# B&R Automation Studio project JXCP_PROFINET_project
Automation Studio 4.9.3.144 SP; technology packages: mappView 5.11.3

## Configuration Config1

CPU X20CP1382, AutomationRuntime A4.73, Build 4.1.2, Safety 0.0, Vc V4.72.0

### Task classes (Cpu.sw)
```
Cyclic#2 (cycle 10000 us, tolerance 10000 us):
  JXCP_Test <- Technology.JXCP_Test.prg
Binaries: udbdef, mvLoader, FWRules, TCData, sysconf, Role, User, iomap, ashwd, asfw, arconfig, ashwac, asnxdb1
Libraries: AsBrMath, rp_funcx, runtime, fileio, astime
```

### Hardware
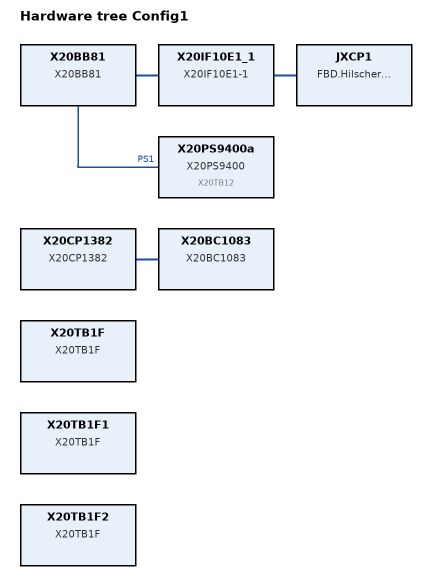
```
JXCP1 : FBD.Hilscher.PNIOGenDevDTM2.JXCP1 v0.0.0.0 (OrderNumber=JXCP1, VendorAddress=jxcp1)  [PN1 -> X20IF10E1_1.IF1]
  DtmId = 32d02dca-1395-427b-a27d-d5b2f34042f0
X20BB81 : X20BB81 v1.0.2.0
X20BC1083 : X20BC1083 v2.11.1.0  [PLK1 -> X20CP1382.IF3 [Cable Type=PowerlinkCable, Length=10, Version=1.0.0.3]; SL -> X20BB81.SL1]
X20CP1382 : X20CP1382 v1.11.0.0  [X1 -> X1.SL; X2 -> X2.SL; X3 -> X3.SL]
  Module X1 (Type=X1, Virtual=true, Version=1.11.0.0)
    Connection (Connector=SS1, TargetModule=X20TB1F, TargetConnector=SS)
    Connection (Connector=SL, TargetModule=X20CP1382, TargetConnector=X1)
  Module X2 (Type=X2, Virtual=true, Version=1.11.0.0)
    Connection (Connector=SS1, TargetModule=X20TB1F1, TargetConnector=SS)
    Connection (Connector=SL, TargetModule=X20CP1382, TargetConnector=X2)
  Module X3 (Type=X3, Virtual=true, Version=1.11.0.0)
    Connection (Connector=SS1, TargetModule=X20TB1F2, TargetConnector=SS)
    Connection (Connector=SL, TargetModule=X20CP1382, TargetConnector=X3)
  Connector IF2:
    ActivateDevice = 1
  Connector IF3:
    DNAConfiguration = manual
  ConfigurationID = JXCP_PROFINET_project_Config1
  Simulation = 1
  SystemTick = 2000
  TaskClassIdleTime = 2000
  Cyclic1Duration = 2000
  Cyclic1Tolerance = 0
  Cyclic2Duration = 10000
  Cyclic2Tolerance = 10000
  ActivateOpcUa = 1
  OpcUaInformationModels_PV_Version = 1
X20IF10E1_1 : X20IF10E1-1 v1.3.0.0  [SS -> X20BB81.SS1]
  Connector IF1:
    DtmRef = FBDIF.Hilscher.PNIOControllerDTM2.NETX 100 RE/PNM
    DtmId = 5926bdb0-bfe7-45dd-88e4-c4368abc1fd1
  ConfigFile = X20IF10E1_1.dtm
  ConfigModule = asnxdb1
  CycleTime = 2000
X20PS9400a : X20PS9400 v1.4.0.0  [SS1 -> X20TB12e.SS; PS -> X20BB81.PS1]
X20TB12e : X20TB12 v1.0.0.0
X20TB1F : X20TB1F v1.0.0.0
X20TB1F1 : X20TB1F v1.0.0.0
X20TB1F2 : X20TB1F v1.0.0.0
```

### IoMap.iom - X20CP1382/IoMap.iom
```iecst
VAR_CONFIG
	::JXCP_Test:jxcp_smc_fb_1.ModuleOK AT %IX."JXCP1".ModuleOk;
	::JXCP_Test.jxcp_smc_fb_1.PROFINET_Mapping_IN.Input_Area[0] AT %IB."JXCP1".Module001_IO_Input001;
	::JXCP_Test.jxcp_smc_fb_1.PROFINET_Mapping_IN.Input_Area[1] AT %IB."JXCP1".Module001_IO_Input002;
	::JXCP_Test.jxcp_smc_fb_1.PROFINET_Mapping_IN.Input_Area[2] AT %IB."JXCP1".Module001_IO_Input003;
	::JXCP_Test.jxcp_smc_fb_1.PROFINET_Mapping_IN.Input_Area[3] AT %IB."JXCP1".Module001_IO_Input004;
	::JXCP_Test.jxcp_smc_fb_1.PROFINET_Mapping_IN.Input_Area[4] AT %IB."JXCP1".Module001_IO_Input005;
	::JXCP_Test.jxcp_smc_fb_1.PROFINET_Mapping_IN.Input_Area[5] AT %IB."JXCP1".Module001_IO_Input006;
	::JXCP_Test.jxcp_smc_fb_1.PROFINET_Mapping_IN.Input_Area[6] AT %IB."JXCP1".Module001_IO_Input007;
	::JXCP_Test.jxcp_smc_fb_1.PROFINET_Mapping_IN.Input_Area[7] AT %IB."JXCP1".Module001_IO_Input008;
	::JXCP_Test.jxcp_smc_fb_1.PROFINET_Mapping_IN.Input_Area[8] AT %IB."JXCP1".Module001_IO_Input009;
	::JXCP_Test.jxcp_smc_fb_1.PROFINET_Mapping_IN.Input_Area[9] AT %IB."JXCP1".Module001_IO_Input010;
	::JXCP_Test.jxcp_smc_fb_1.PROFINET_Mapping_IN.Input_Area[10] AT %IB."JXCP1".Module001_IO_Input011;
	::JXCP_Test.jxcp_smc_fb_1.PROFINET_Mapping_IN.Input_Area[11] AT %IB."JXCP1".Module001_IO_Input012;
	::JXCP_Test.jxcp_smc_fb_1.PROFINET_Mapping_IN.Input_Area[12] AT %IB."JXCP1".Module001_IO_Input013;
	::JXCP_Test.jxcp_smc_fb_1.PROFINET_Mapping_IN.Input_Area[13] AT %IB."JXCP1".Module001_IO_Input014;
	::JXCP_Test.jxcp_smc_fb_1.PROFINET_Mapping_IN.Input_Area[14] AT %IB."JXCP1".Module001_IO_Input015;
	::JXCP_Test.jxcp_smc_fb_1.PROFINET_Mapping_IN.Input_Area[15] AT %IB."JXCP1".Module001_IO_Input016;
	::JXCP_Test.jxcp_smc_fb_1.PROFINET_Mapping_IN.Input_Area[16] AT %IB."JXCP1".Module001_IO_Input017;
	::JXCP_Test.jxcp_smc_fb_1.PROFINET_Mapping_IN.Input_Area[17] AT %IB."JXCP1".Module001_IO_Input018;
	::JXCP_Test.jxcp_smc_fb_1.PROFINET_Mapping_IN.Input_Area[18] AT %IB."JXCP1".Module001_IO_Input019;
	::JXCP_Test.jxcp_smc_fb_1.PROFINET_Mapping_IN.Input_Area[19] AT %IB."JXCP1".Module001_IO_Input020;
	::JXCP_Test:jxcp_smc_fb_1.PROFINET_Mapping_OUT.Output_Area[0] AT %QB."JXCP1".Module002_IO_Output001;
	::JXCP_Test:jxcp_smc_fb_1.PROFINET_Mapping_OUT.Output_Area[1] AT %QB."JXCP1".Module002_IO_Output002;
	::JXCP_Test:jxcp_smc_fb_1.PROFINET_Mapping_OUT.Output_Area[2] AT %QB."JXCP1".Module002_IO_Output003;
	::JXCP_Test:jxcp_smc_fb_1.PROFINET_Mapping_OUT.Output_Area[3] AT %QB."JXCP1".Module002_IO_Output004;
	::JXCP_Test:jxcp_smc_fb_1.PROFINET_Mapping_OUT.Output_Area[4] AT %QB."JXCP1".Module002_IO_Output005;
	::JXCP_Test:jxcp_smc_fb_1.PROFINET_Mapping_OUT.Output_Area[5] AT %QB."JXCP1".Module002_IO_Output006;
	::JXCP_Test:jxcp_smc_fb_1.PROFINET_Mapping_OUT.Output_Area[6] AT %QB."JXCP1".Module002_IO_Output007;
	::JXCP_Test:jxcp_smc_fb_1.PROFINET_Mapping_OUT.Output_Area[7] AT %QB."JXCP1".Module002_IO_Output008;
	::JXCP_Test:jxcp_smc_fb_1.PROFINET_Mapping_OUT.Output_Area[8] AT %QB."JXCP1".Module002_IO_Output009;
	::JXCP_Test:jxcp_smc_fb_1.PROFINET_Mapping_OUT.Output_Area[9] AT %QB."JXCP1".Module002_IO_Output010;
	::JXCP_Test:jxcp_smc_fb_1.PROFINET_Mapping_OUT.Output_Area[10] AT %QB."JXCP1".Module002_IO_Output011;
	::JXCP_Test:jxcp_smc_fb_1.PROFINET_Mapping_OUT.Output_Area[11] AT %QB."JXCP1".Module002_IO_Output012;
	::JXCP_Test:jxcp_smc_fb_1.PROFINET_Mapping_OUT.Output_Area[12] AT %QB."JXCP1".Module002_IO_Output013;
	::JXCP_Test:jxcp_smc_fb_1.PROFINET_Mapping_OUT.Output_Area[13] AT %QB."JXCP1".Module002_IO_Output014;
	::JXCP_Test:jxcp_smc_fb_1.PROFINET_Mapping_OUT.Output_Area[14] AT %QB."JXCP1".Module002_IO_Output015;
	::JXCP_Test:jxcp_smc_fb_1.PROFINET_Mapping_OUT.Output_Area[15] AT %QB."JXCP1".Module002_IO_Output016;
	::JXCP_Test:jxcp_smc_fb_1.PROFINET_Mapping_OUT.Output_Area[16] AT %QB."JXCP1".Module002_IO_Output017;
	::JXCP_Test:jxcp_smc_fb_1.PROFINET_Mapping_OUT.Output_Area[17] AT %QB."JXCP1".Module002_IO_Output018;
	::JXCP_Test:jxcp_smc_fb_1.PROFINET_Mapping_OUT.Output_Area[18] AT %QB."JXCP1".Module002_IO_Output019;
	::JXCP_Test:jxcp_smc_fb_1.PROFINET_Mapping_OUT.Output_Area[19] AT %QB."JXCP1".Module002_IO_Output020;
	::JXCP_Test:jxcp_smc_fb_1.PROFINET_Mapping_OUT.Output_Area[20] AT %QB."JXCP1".Module002_IO_Output021;
	::JXCP_Test:jxcp_smc_fb_1.PROFINET_Mapping_OUT.Output_Area[21] AT %QB."JXCP1".Module002_IO_Output022;
	::JXCP_Test:jxcp_smc_fb_1.PROFINET_Mapping_OUT.Output_Area[22] AT %QB."JXCP1".Module002_IO_Output023;
	::JXCP_Test:jxcp_smc_fb_1.PROFINET_Mapping_OUT.Output_Area[23] AT %QB."JXCP1".Module002_IO_Output024;
	::JXCP_Test:jxcp_smc_fb_1.PROFINET_Mapping_OUT.Output_Area[24] AT %QB."JXCP1".Module002_IO_Output025;
	::JXCP_Test:jxcp_smc_fb_1.PROFINET_Mapping_OUT.Output_Area[25] AT %QB."JXCP1".Module002_IO_Output026;
	::JXCP_Test:jxcp_smc_fb_1.PROFINET_Mapping_OUT.Output_Area[26] AT %QB."JXCP1".Module002_IO_Output027;
	::JXCP_Test:jxcp_smc_fb_1.PROFINET_Mapping_OUT.Output_Area[27] AT %QB."JXCP1".Module002_IO_Output028;
	::JXCP_Test:jxcp_smc_fb_1.PROFINET_Mapping_OUT.Output_Area[28] AT %QB."JXCP1".Module002_IO_Output029;
	::JXCP_Test:jxcp_smc_fb_1.PROFINET_Mapping_OUT.Output_Area[29] AT %QB."JXCP1".Module002_IO_Output030;
	::JXCP_Test:jxcp_smc_fb_1.PROFINET_Mapping_OUT.Output_Area[30] AT %QB."JXCP1".Module002_IO_Output031;
	::JXCP_Test:jxcp_smc_fb_1.PROFINET_Mapping_OUT.Output_Area[31] AT %QB."JXCP1".Module002_IO_Output032;
	::JXCP_Test:jxcp_smc_fb_1.PROFINET_Mapping_OUT.Output_Area[32] AT %QB."JXCP1".Module002_IO_Output033;
	::JXCP_Test:jxcp_smc_fb_1.PROFINET_Mapping_OUT.Output_Area[33] AT %QB."JXCP1".Module002_IO_Output034;
	::JXCP_Test:jxcp_smc_fb_1.PROFINET_Mapping_OUT.Output_Area[34] AT %QB."JXCP1".Module002_IO_Output035;
	::JXCP_Test:jxcp_smc_fb_1.PROFINET_Mapping_OUT.Output_Area[35] AT %QB."JXCP1".Module002_IO_Output036;
END_VAR
```

## Logical view

Binary libraries used (declarations not repeated): operator, runtime, astime, AsIecCon, AsBrMath

### Global.typ - Global data types
```iecst
TYPE
	jxcp_mv_alarm_str : 	STRUCT
		Alarm_1 : USINT;
		Alarm_1_img : BOOL;
		Alarm_2 : USINT;
		Alarm_2_img : BOOL;
		Alarm_3 : USINT;
		Alarm_3_img : BOOL;
		Alarm_4 : USINT;
		Alarm_4_img : BOOL;
	END_STRUCT;
	jxcp_mv_get_param_str : 	STRUCT
		Position : LREAL;
		Speed : LREAL;
		Force : LREAL;
		In_Pos : BOOL;
	END_STRUCT;
	jxcp_data_mv_str : 	STRUCT
		Power : BOOL;
		Home : BOOL;
		isHome : BOOL;
		PowerOn : BOOL;
		Control : jxcp_mv_control_str;
		Write_Parameters : jxcp_mv_set_param_str;
		Read_Parameters : jxcp_mv_get_param_str;
		Alarm : jxcp_mv_alarm_str;
		Reset_Alarm : BOOL;
	END_STRUCT;
	jxcp_mv_cm_str : 	STRUCT
		Start : BOOL;
		Stop : BOOL;
		Default_Param : BOOL;
	END_STRUCT;
	jxcp_mv_control_str : 	STRUCT
		Jog_pos : BOOL;
		Jog_neg : BOOL;
		Cycle_Mode : jxcp_mv_cm_str;
	END_STRUCT;
	jxcp_mv_set_param_str : 	STRUCT
		Position : LREAL;
		Speed : LREAL;
		Acceleration : LREAL;
		Deceleration : LREAL;
	END_STRUCT;
END_TYPE
```

### Global.var - Global variables
```iecst
VAR
	jxcp_data_mv : jxcp_data_mv_str;
END_VAR
```

### Package Logical/Libraries - Global libraries

### Library Logical/Libraries/rp_funcx (ANSIC)

#### Types.typ - Exported data types
```iecst
TYPE
	profinet_aux_m_str : 	STRUCT
		IN_Aux : profinet_aux_in_str;
		OUT_Aux : profinet_aux_out_str;
	END_STRUCT;
	profinet_aux_out_str : 	STRUCT
		BYTE_0 : ARRAY[0..5]OF BOOL;
		BYTE_1 : ARRAY[0..7]OF BOOL;
		BYTE_2 : BOOL;
	END_STRUCT;
	jxcp_main_read_enum :
		(
		JXCP_R_INITIALIZATION_STATE := 0,
		JXCP_R_RW_STATE := 10,
		JXCP_R_ERROR_MODE_STATE := 20
		);
	profinet_aux_in_str : 	STRUCT
		BYTE_0 : ARRAY[0..5]OF BOOL;
		BYTE_1 : ARRAY[0..7]OF BOOL;
		BYTE_2 : ARRAY[0..7]OF BOOL;
		BYTE_3 : ARRAY[0..7]OF BOOL;
	END_STRUCT;
	jxcp_main_enum :
		(
		JXCP_INITIALIZATION_STATE := 0,
		JXCP_WAIT_STATE := 10,
		JXCP_CYCLE_MODE_STATE := 20,
		JXCP_ALARM_MODE_STATE := 30,
		JXCP_ERROR_MODE_STATE := 40
		);
	set_param_mode_enum :
		(
		CYCLE_MOVE_MODE := 0
		);
	internal_param_str : 	STRUCT
		actual_state : jxcp_main_enum;
		before_state : jxcp_main_enum;
		actual_r_state : jxcp_main_read_enum;
		before_r_state : jxcp_main_read_enum;
		Profinet : profinet_aux_m_str;
	END_STRUCT;
	set_param_str : 	STRUCT
		Start : BOOL;
		Stop : BOOL;
		Mode : set_param_mode_enum;
		Boundary : boundary_str;
	END_STRUCT;
	byte_3_in_str : 	STRUCT
		Deceleration : BOOL;
		Pushing_Force : BOOL;
		Trigger_LV : BOOL;
		Pushing_Speed : BOOL;
		Moving_Force : BOOL;
		Area_out_1 : BOOL;
		Area_out_2 : BOOL;
		IN_Pos_Tolerance : BOOL;
	END_STRUCT;
	byte_2_in_str : 	STRUCT
		Speed_Restriction : BOOL;
		Movement_Mode : BOOL;
		Speed : BOOL;
		Position : BOOL;
		Acceleration : BOOL;
	END_STRUCT;
	byte_1_in_str : 	STRUCT
		HOLD : BOOL;
		SVON : BOOL;
		DRIVE : BOOL;
		RESET : BOOL;
		SETUP : BOOL;
		JOG_Neg : BOOL;
		JOG_Pos : BOOL;
		FLHGT : BOOL;
	END_STRUCT;
	byte_0_in_str : 	STRUCT
		IN_0 : BOOL;
		IN_1 : BOOL;
		IN_2 : BOOL;
		IN_3 : BOOL;
		IN_4 : BOOL;
		IN_5 : BOOL;
	END_STRUCT;
	movement_mode_str : 	STRUCT
		Absolute : BOOL;
		Relative : BOOL;
	END_STRUCT;
	alarm_str : 	STRUCT
		Alarm_1 : USINT;
		Alarm_2 : USINT;
		Alarm_3 : USINT;
		Alarm_4 : USINT;
	END_STRUCT;
	byte_2_str : 	STRUCT
		READY : BOOL;
	END_STRUCT;
	byte_1_str : 	STRUCT
		BUSY : BOOL;
		SVRE : BOOL;
		SETON : BOOL;
		INP : BOOL;
		AREA : BOOL;
		WAREA : BOOL;
		ESTOP : BOOL;
		ALARM : BOOL;
	END_STRUCT;
	byte_0_str : 	STRUCT
		OUT_0 : BOOL;
		OUT_1 : BOOL;
		OUT_2 : BOOL;
		OUT_3 : BOOL;
		OUT_4 : BOOL;
		OUT_5 : BOOL;
	END_STRUCT;
	jxcp_input_str : 	STRUCT
		BYTE_0 : byte_0_in_str;
		BYTE_1 : byte_1_in_str;
		BYTE_2 : byte_2_in_str;
		BYTE_3 : byte_3_in_str;
		Start_Flag : BOOL;
		Movement_Mode : movement_mode_str;
		Speed : LREAL;
		Position : LREAL;
		Acceleration : LREAL;
		Deceleration : LREAL;
		Pushing_Force : LREAL;
		Trigger_LV : LREAL;
		Pushing_Speed : LREAL;
		Moving_Force : LREAL;
		AREA_1 : LREAL;
		AREA_2 : LREAL;
		IN_Position : LREAL;
	END_STRUCT;
	jxcp_output_str : 	STRUCT
		BYTE_0 : byte_0_str;
		BYTE_1 : byte_1_str;
		BYTE_2 : byte_2_str;
		Current_Position : LREAL;
		Current_Speed : LREAL;
		Current_Pushing_Force : LREAL;
		Target_Position : LREAL;
		Warning : alarm_str;
	END_STRUCT;
	profinet_mapping_out_str : 	STRUCT
		Output_Area : ARRAY[0..35]OF USINT;
	END_STRUCT;
	profinet_mapping_in_str : 	STRUCT
		Input_Area : ARRAY[0..19]OF USINT;
	END_STRUCT;
	boundary_mm_str : 	STRUCT
		max : LREAL;
		min : LREAL;
	END_STRUCT;
	boundary_str : 	STRUCT
		Position : boundary_mm_str;
		Speed : boundary_mm_str;
		Acceleration : boundary_mm_str;
		Deceleration : boundary_mm_str;
	END_STRUCT;
END_TYPE
```

#### rp_funcx.fun - Exported functions and function blocks
```iecst
FUNCTION_BLOCK dec_to_multiple_usint
	VAR_INPUT
		Count_of_VAR : USINT;
		Decimal : LREAL;
	END_VAR
	VAR_OUTPUT
		Result_USINT_1 : USINT;
		Result_USINT_2 : USINT;
		Result_USINT_3 : USINT;
		Result_USINT_4 : USINT;
	END_VAR
END_FUNCTION_BLOCK

FUNCTION_BLOCK multiplne_usint_to_dec
	VAR_INPUT
		Count_of_VAR : USINT;
		USINT_1 : USINT;
		USINT_2 : USINT;
		USINT_3 : USINT;
		USINT_4 : USINT;
	END_VAR
	VAR_OUTPUT
		Result_Decimal : LREAL;
	END_VAR
END_FUNCTION_BLOCK

{REDUND_ERROR} FUNCTION_BLOCK jxcp_smc_fb (*TODO: Add your comment here*) (*$GROUP=User,$CAT=User,$GROUPICON=User.png,$CATICON=User.png*)
	VAR_INPUT
		Enable : {REDUND_UNREPLICABLE} BOOL;
		ModuleOK : BOOL;
		PROFINET_Mapping_IN : {REDUND_UNREPLICABLE} profinet_mapping_in_str;
		Input : jxcp_input_str;
		Set_Parameters : set_param_str;
	END_VAR
	VAR_OUTPUT
		Active : BOOL;
		PROFINET_Mapping_OUT : profinet_mapping_out_str;
		Output : jxcp_output_str;
	END_VAR
	VAR
		Internal : internal_param_str;
	END_VAR
END_FUNCTION_BLOCK
```

#### jxcp_smc_fb.c
```c
// ************************************************************************************************************************************ //
// Title: JXCP1 (SMC) - Control {PROFINET}
// Autor: Roman Parak
// Date : 8.5.2020
// Email: Roman.Parak@outlook.com
// ************************************************************************************************************************************ //

// ************************************************************************************************************************************ //
// -------------------------------------------------------------  LIBRARIES ----------------------------------------------------------- //
// ************************************************************************************************************************************ //
#include <bur/plctypes.h>
#include <stdio.h>
#include <stdlib.h>
#include <math.h>

#ifdef __cplusplus
	extern "C"
	{
#endif
#include "rp_funcx.h"
#ifdef __cplusplus
	};
#endif

// ************************************************************************************************************************************ //
// -------------------------------------------------------------  DECLARATIONS -------------------------------------------------------- //
// ************************************************************************************************************************************ //
// INITIALIZATION // RESET //
void initialization_jxcp(struct jxcp_smc_fb* jxcp_s);

// INITIALIZATION // AUX. FCE. Convert Binary to Decimal //
DINT convert_bin_to_dec(LREAL n);

// ************************************************************************************************************************************ //
// --------------------------------------------------------------  MAIN --------------------------------------------------------------- //
// ************************************************************************************************************************************ //
void jxcp_smc_fb(struct jxcp_smc_fb* jxcp_s)
{
	// *********************************************************//
	// ---------------- INITIALIZATION  ----------------------- //
	// *********************************************************//
	if(jxcp_s->Enable != 1){
		initialization_jxcp(jxcp_s);
	}

	// declaration index {all cycles)
	int i, i_w;

	// Read {Multiple USINT to Decimal -> Function Block}
	struct multiple_usint_to_dec m_u2d_cP; // Current Position
	struct multiple_usint_to_dec m_u2d_cS; // Current Speed
	struct multiple_usint_to_dec m_u2d_cPF; // Current Pushing Force
	struct multiple_usint_to_dec m_u2d_TP; // Target Position

	// Write {Decimal to multiple USINT -> Function Block}
	struct dec_to_multiple_usint dec2u_m_S; // Speed
	struct dec_to_multiple_usint dec2u_m_P; // Position
	struct dec_to_multiple_usint dec2u_m_Acc; // Acceleration
	struct dec_to_multiple_usint dec2u_m_Dec; // Deceleration
	struct dec_to_multiple_usint dec2u_m_PF; // Pushing Force
	struct dec_to_multiple_usint dec2u_m_TLV; // Trigger LV
	struct dec_to_multiple_usint dec2u_m_PS; // Pushing Speed
	struct dec_to_multiple_usint dec2u_m_MF; // Moving FOrce
	struct dec_to_multiple_usint dec2u_m_AR1; // Area 1
	struct dec_to_multiple_usint dec2u_m_AR2; // Area 2
	struct dec_to_multiple_usint dec2u_m_IN_P; // IN Position

	// ******************************************************************************************************************//
	// --------------------------------------------- JXCP MAIN STATE  -------------------------------------------------- //
	// ******************************************************************************************************************//
	switch(jxcp_s->Internal.actual_state){
		case JXCP_INITIALIZATION_STATE:
			{
				/*************************************** INITIALIZATION STATE ******************************************/
				jxcp_s->Internal.before_state = JXCP_INITIALIZATION_STATE;
				// Profinet Module -> OK
				if(jxcp_s->ModuleOK == 1){
					// Set FB -> Active 1
					jxcp_s->Active = 1;
					// Change State -> Wait
					jxcp_s->Internal.actual_state = JXCP_WAIT_STATE;
				}
			}
			break;
		case JXCP_WAIT_STATE:
			{
				/*************************************** WAIT STATE ******************************************/
				jxcp_s->Internal.before_state = JXCP_WAIT_STATE;

				jxcp_s->Set_Parameters.Stop = 0;

				// *************** Start Mode *************** //
				if(jxcp_s->Set_Parameters.Start == 1){
					if(jxcp_s->Set_Parameters.Mode == NORMAL_MOVE_MODE){
						// Normal Mode
						jxcp_s->Internal.actual_state = JXCP_NORMAL_MODE_STATE;
					}else if(jxcp_s->Set_Parameters.Mode == CYCLE_MOVE_MODE){
						// Write Byte 2 { SET - 1 }
						jxcp_s->Input.BYTE_2.Speed_Restriction = 1;
						jxcp_s->Input.BYTE_2.Movement_Mode     = 1;
						jxcp_s->Input.BYTE_2.Speed             = 1;
						jxcp_s->Input.BYTE_2.Position          = 1;
						jxcp_s->Input.BYTE_2.Acceleration      = 1;
						// Write Byte 3 { SET - 1 }
						jxcp_s->Input.BYTE_3.Deceleration      = 1;
						jxcp_s->Input.BYTE_3.Pushing_Force     = 1;
						jxcp_s->Input.BYTE_3.Trigger_LV        = 1;
						jxcp_s->Input.BYTE_3.Pushing_Speed     = 1;
						jxcp_s->Input.BYTE_3.Moving_Force      = 1;
						jxcp_s->Input.BYTE_3.Area_out_1        = 1;
						jxcp_s->Input.BYTE_3.Area_out_2        = 1;
						jxcp_s->Input.BYTE_3.IN_Pos_Tolerance  = 1;
						// Cycle Mode
						jxcp_s->Internal.actual_state = JXCP_CYCLE_MODE_STATE;
					}
				}

				// Module OK = 0 -> Error State
				if(jxcp_s->ModuleOK != 1){
					// Set FB -> Active 0
					jxcp_s->Active = 0;
					// Change State -> Error
					jxcp_s->Internal.actual_state = JXCP_ERROR_MODE_STATE;
				}
			}
			break;
		case JXCP_NORMAL_MODE_STATE:
			{
				/*************************************** NORMAL MODE STATE ******************************************/
				jxcp_s->Internal.before_state = JXCP_NORMAL_MODE_STATE;

				// *************** Stop Actual Mode *************** //
				if(jxcp_s->Set_Parameters.Stop == 1){
					jxcp_s->Set_Parameters.Start = 0;
					// Change State -> Initialization
					jxcp_s->Internal.actual_state = JXCP_WAIT_STATE;
				}

				// Module OK = 0 -> Error State
				if(jxcp_s->ModuleOK != 1){
					// Set FB -> Active 0
					jxcp_s->Active = 0;
					// Change State -> Error
					jxcp_s->Internal.actual_state = JXCP_ERROR_MODE_STATE;
				}
			}
			break;
		case JXCP_CYCLE_MODE_STATE:
			{
				/*************************************** CYCLE MODE STATE ******************************************/
				jxcp_s->Internal.before_state = JXCP_CYCLE_MODE_STATE;

				// Start Cycle Mode -> JXCP1 command
				jxcp_s->Input.Start_Flag 			 = 1;
				// Movement Mode - Absolute
				jxcp_s->Input.Movement_Mode.Absolute = 1;

				/*************************************************************************/
				/*************** Calculation  DEC. TO MULTIPLE USINT *********************/
				/*************************************************************************/

				// *************** Speed *************** //
				// Number of Variables (USINT)
				dec2u_m_S.Count_of_VAR = 2;
				// Boundary Condition
				if(jxcp_s->Input.Speed > jxcp_s->Set_Parameters.Boundary.Speed.max){
					dec2u_m_S.Decimal = jxcp_s->Set_Parameters.Boundary.Speed.max;
				}else if(jxcp_s->Input.Speed < jxcp_s->Set_Parameters.Boundary.Speed.min){
					dec2u_m_S.Decimal = jxcp_s->Set_Parameters.Boundary.Speed.min;
				}else{
					dec2u_m_S.Decimal = jxcp_s->Input.Speed;
				}
				// Call Function Block (Decimal to Multiple USINT)
				dec_to_multiple_usint(&dec2u_m_S);
				// Result (Write -> PROFINET Module)
				jxcp_s->PROFINET_Mapping_OUT.Output_Area[6] = dec2u_m_S.Result_USINT_1;
				jxcp_s->PROFINET_Mapping_OUT.Output_Area[7] = dec2u_m_S.Result_USINT_2;

				// *************** Position *************** //
				// Number of Variables (USINT)
				dec2u_m_P.Count_of_VAR = 4;
				// Boundary Condition
				if(jxcp_s->Input.Position > jxcp_s->Set_Parameters.Boundary.Position.max){
					dec2u_m_P.Decimal = jxcp_s->Set_Parameters.Boundary.Position.max;
				}else if(jxcp_s->Input.Position < jxcp_s->Set_Parameters.Boundary.Position.min){
					dec2u_m_P.Decimal = jxcp_s->Set_Parameters.Boundary.Position.min;
				}else{
					dec2u_m_P.Decimal = jxcp_s->Input.Position;
				}
				// Call Function Block (Decimal to Multiple USINT)
				dec_to_multiple_usint(&dec2u_m_P);
				// Result (Write -> PROFINET Module)
				jxcp_s->PROFINET_Mapping_OUT.Output_Area[8] = dec2u_m_P.Result_USINT_1;
				jxcp_s->PROFINET_Mapping_OUT.Output_Area[9] = dec2u_m_P.Result_USINT_2;
				jxcp_s->PROFINET_Mapping_OUT.Output_Area[10] = dec2u_m_P.Result_USINT_3;
				jxcp_s->PROFINET_Mapping_OUT.Output_Area[11] = dec2u_m_P.Result_USINT_4;

				// *************** Acceleration *************** //
				// Number of Variables (USINT)
				dec2u_m_Acc.Count_of_VAR = 2;
				// Boundary Condition
				if(jxcp_s->Input.Acceleration > jxcp_s->Set_Parameters.Boundary.Acceleration.max){
					dec2u_m_Acc.Decimal = jxcp_s->Set_Parameters.Boundary.Acceleration.max;
				}else if(jxcp_s->Input.Acceleration < jxcp_s->Set_Parameters.Boundary.Acceleration.min){
					dec2u_m_Acc.Decimal = jxcp_s->Set_Parameters.Boundary.Acceleration.min;
				}else{
					dec2u_m_Acc.Decimal = jxcp_s->Input.Acceleration;
				}
				// Call Function Block (Decimal to Multiple USINT)
				dec_to_multiple_usint(&dec2u_m_Acc);
				// Result (Write -> PROFINET Module)
				jxcp_s->PROFINET_Mapping_OUT.Output_Area[12] = dec2u_m_Acc.Result_USINT_1;
				jxcp_s->PROFINET_Mapping_OUT.Output_Area[13] = dec2u_m_Acc.Result_USINT_2;

				// *************** Deceleration *************** //
				// Number of Variables (USINT)
				dec2u_m_Dec.Count_of_VAR = 2;
				// Boundary Condition
				if(jxcp_s->Input.Deceleration > jxcp_s->Set_Parameters.Boundary.Deceleration.max){
					dec2u_m_Dec.Decimal = jxcp_s->Set_Parameters.Boundary.Deceleration.max;
				}else if(jxcp_s->Input.Deceleration < jxcp_s->Set_Parameters.Boundary.Deceleration.min){
					dec2u_m_Dec.Decimal = jxcp_s->Set_Parameters.Boundary.Deceleration.min;
				}else{
					dec2u_m_Dec.Decimal = jxcp_s->Input.Deceleration;
				}
				// Call Function Block (Decimal to Multiple USINT)
				dec_to_multiple_usint(&dec2u_m_Dec);
				// Result (Write -> PROFINET Module)
				jxcp_s->PROFINET_Mapping_OUT.Output_Area[14] = dec2u_m_Dec.Result_USINT_1;
				jxcp_s->PROFINET_Mapping_OUT.Output_Area[15] = dec2u_m_Dec.Result_USINT_2;

				// *************** Pushing Force *************** //
				// Number of Variables (USINT)
				dec2u_m_PF.Count_of_VAR = 2;
				// Boundary Condition (NO)
				dec2u_m_PF.Decimal = jxcp_s->Input.Pushing_Force;
				// Call Function Block (Decimal to Multiple USINT)
				dec_to_multiple_usint(&dec2u_m_PF);
				// Result (Write -> PROFINET Module)
				jxcp_s->PROFINET_Mapping_OUT.Output_Area[16] = dec2u_m_PF.Result_USINT_1;
				jxcp_s->PROFINET_Mapping_OUT.Output_Area[17] = dec2u_m_PF.Result_USINT_2;

				// *************** Trigger LV *************** //
				// Number of Variables (USINT)
				dec2u_m_TLV.Count_of_VAR = 2;
				// Boundary Condition (NO)
				dec2u_m_TLV.Decimal = jxcp_s->Input.Trigger_LV;
				// Call Function Block (Decimal to Multiple USINT)
				dec_to_multiple_usint(&dec2u_m_TLV);
				// Result (Write -> PROFINET Module)
				jxcp_s->PROFINET_Mapping_OUT.Output_Area[18] = dec2u_m_TLV.Result_USINT_1;
				jxcp_s->PROFINET_Mapping_OUT.Output_Area[19] = dec2u_m_TLV.Result_USINT_2;

				// *************** Pushing Speed *************** //
				// Number of Variables (USINT)
				dec2u_m_PS.Count_of_VAR = 2;
				// Boundary Condition (NO)
				dec2u_m_PS.Decimal = jxcp_s->Input.Pushing_Speed;
				// Call Function Block (Decimal to Multiple USINT)
				dec_to_multiple_usint(&dec2u_m_PS);
				// Result (Write -> PROFINET Module)
				jxcp_s->PROFINET_Mapping_OUT.Output_Area[20] = dec2u_m_PS.Result_USINT_1;
				jxcp_s->PROFINET_Mapping_OUT.Output_Area[21] = dec2u_m_PS.Result_USINT_2;

				// *************** Moving Force *************** //
				// Number of Variables (USINT)
				dec2u_m_MF.Count_of_VAR = 2;
				// Boundary Condition (NO)
				dec2u_m_MF.Decimal = jxcp_s->Input.Moving_Force;
				// Call Function Block (Decimal to Multiple USINT)
				dec_to_multiple_usint(&dec2u_m_MF);
				// Result (Write -> PROFINET Module)
				jxcp_s->PROFINET_Mapping_OUT.Output_Area[22] = dec2u_m_MF.Result_USINT_1;
				jxcp_s->PROFINET_Mapping_OUT.Output_Area[23] = dec2u_m_MF.Result_USINT_2;

				// *************** Area 1 *************** //
				// Number of Variables (USINT)
				dec2u_m_AR1.Count_of_VAR = 4;
				// Boundary Condition (NO)
				dec2u_m_AR1.Decimal = jxcp_s->Input.AREA_1;
				// Call Function Block (Decimal to Multiple USINT)
				dec_to_multiple_usint(&dec2u_m_AR1);
				// Result (Write -> PROFINET Module)
				jxcp_s->PROFINET_Mapping_OUT.Output_Area[24] = dec2u_m_AR1.Result_USINT_1;
				jxcp_s->PROFINET_Mapping_OUT.Output_Area[25] = dec2u_m_AR1.Result_USINT_2;
				jxcp_s->PROFINET_Mapping_OUT.Output_Area[26] = dec2u_m_AR1.Result_USINT_3;
				jxcp_s->PROFINET_Mapping_OUT.Output_Area[27] = dec2u_m_AR1.Result_USINT_4;

				// *************** Area 2 *************** //
				// Number of Variables (USINT)
				dec2u_m_AR2.Count_of_VAR = 4;
				// Boundary Condition (NO)
				dec2u_m_AR2.Decimal = jxcp_s->Input.AREA_2;
				// Call Function Block (Decimal to Multiple USINT)
				dec_to_multiple_usint(&dec2u_m_AR2);
				// Result (Write -> PROFINET Module)
				jxcp_s->PROFINET_Mapping_OUT.Output_Area[28] = dec2u_m_AR2.Result_USINT_1;
				jxcp_s->PROFINET_Mapping_OUT.Output_Area[29] = dec2u_m_AR2.Result_USINT_2;
				jxcp_s->PROFINET_Mapping_OUT.Output_Area[30] = dec2u_m_AR2.Result_USINT_3;
				jxcp_s->PROFINET_Mapping_OUT.Output_Area[31] = dec2u_m_AR2.Result_USINT_4;

				// *************** In-Position *************** //
				// Number of Variables (USINT)
				dec2u_m_IN_P.Count_of_VAR = 4;
				// Boundary Condition (NO)
				dec2u_m_IN_P.Decimal = jxcp_s->Input.IN_Position;
				// Call Function Block (Decimal to Multiple USINT)
				dec_to_multiple_usint(&dec2u_m_IN_P);
				// Result (Write -> PROFINET Module)
				jxcp_s->PROFINET_Mapping_OUT.Output_Area[32] = dec2u_m_IN_P.Result_USINT_1;
				jxcp_s->PROFINET_Mapping_OUT.Output_Area[33] = dec2u_m_IN_P.Result_USINT_2;
				jxcp_s->PROFINET_Mapping_OUT.Output_Area[34] = dec2u_m_IN_P.Result_USINT_3;
				jxcp_s->PROFINET_Mapping_OUT.Output_Area[35] = dec2u_m_IN_P.Result_USINT_4;

				// *************** Stop Actual Mode *************** //
				if(jxcp_s->Set_Parameters.Stop == 1){
					jxcp_s->Set_Parameters.Start = 0;
					// Write Byte 4 { SET - 0 }
					jxcp_s->Input.Start_Flag 			   = 0;
					// Write Byte 2 { SET - 0 }
					jxcp_s->Input.BYTE_2.Speed_Restriction = 0;
					jxcp_s->Input.BYTE_2.Movement_Mode     = 0;
					jxcp_s->Input.BYTE_2.Speed             = 0;
					jxcp_s->Input.BYTE_2.Position          = 0;
					jxcp_s->Input.BYTE_2.Acceleration      = 0;
					// Write Byte 3 { SET - 0 }
					jxcp_s->Input.BYTE_3.Deceleration      = 0;
					jxcp_s->Input.BYTE_3.Pushing_Force     = 0;
					jxcp_s->Input.BYTE_3.Trigger_LV        = 0;
					jxcp_s->Input.BYTE_3.Pushing_Speed     = 0;
					jxcp_s->Input.BYTE_3.Moving_Force      = 0;
					jxcp_s->Input.BYTE_3.Area_out_1        = 0;
					jxcp_s->Input.BYTE_3.Area_out_2        = 0;
					jxcp_s->Input.BYTE_3.IN_Pos_Tolerance  = 0;
					// Change State -> Initialization
					jxcp_s->Internal.actual_state = JXCP_WAIT_STATE;
				}

				// Module OK = 0 -> Error State
				if(jxcp_s->ModuleOK != 1){
					// Set FB -> Active 0
					jxcp_s->Active = 0;
					// Change State -> Error
					jxcp_s->Internal.actual_state = JXCP_ERROR_MODE_STATE;
				}
			}
			break;
		case JXCP_ALARM_MODE_STATE:
			{
				/*************************************** ALARM STATE ******************************************/
				jxcp_s->Internal.before_state = JXCP_ALARM_MODE_STATE;

				// Module OK = 0 -> Error State
				if(jxcp_s->ModuleOK != 1){
					// Set FB -> Active 0
					jxcp_s->Active = 0;
					// Change State -> Error
					jxcp_s->Internal.actual_state = JXCP_ERROR_MODE_STATE;
				}
			}
			break;
		case JXCP_ERROR_MODE_STATE:
			{
				/*************************************** ERROR STATE ******************************************/
				// Profinet Module -> OK
				if(jxcp_s->ModuleOK == 1){
					// Set FB -> Active 1
					jxcp_s->Active = 1;
					// Change State -> before state (before the error)
					jxcp_s->Internal.actual_state = jxcp_s->Internal.before_state;
				}
			}
			break;
	} // end switch

	// ******************************************************************************************************************//
	// ---------------------------------------------------- JXCP R/W STATE  -------------------------------------------- //
	// ******************************************************************************************************************//
	switch(jxcp_s->Internal.actual_r_state){
		case JXCP_R_INITIALIZATION_STATE:
			{
				/*************************************** INITIALIZATION STATE ******************************************/
				jxcp_s->Internal.before_r_state = JXCP_R_INITIALIZATION_STATE;
				// Profinet Module -> OK
				if(jxcp_s->ModuleOK == 1){
					// Set FB -> Active
					jxcp_s->Active = 1;
					// Change State -> Read/Write
					jxcp_s->Internal.actual_r_state = JXCP_R_RW_STATE;
				}
			}
			break;
		case JXCP_R_RW_STATE:
			{
				/*************************************** READ/WRITE STATE ******************************************/
				jxcp_s->Internal.before_r_state = JXCP_R_RW_STATE;

				// ************************************************************************ //
				// ********************************* READ ********************************* //
				// ************************************************************************ //

				// *************** Byte 0 *************** //
				// Create aux. variable
				USINT aux_get_byte_0;
				// Read Profinet Var.
				aux_get_byte_0 = jxcp_s->PROFINET_Mapping_IN.Input_Area[0];
				// Calculation Boolean (True/False) array (Byte 0)
				for(i = 0; i < (int)(sizeof(jxcp_s->Internal.Profinet.OUT_Aux.BYTE_0)/sizeof(jxcp_s->Internal.Profinet.OUT_Aux.BYTE_0[0])); i++){
					if(aux_get_byte_0 > 0){
						jxcp_s->Internal.Profinet.OUT_Aux.BYTE_0[i] = aux_get_byte_0 % 2;
						aux_get_byte_0 = aux_get_byte_0/2;
					}else{
						jxcp_s->Internal.Profinet.OUT_Aux.BYTE_0[i] = 0;
					}
				}

				// *************** Byte 1 *************** //
				// Create aux. variable
				USINT aux_get_byte_1;
				// Read Profinet Var.
				aux_get_byte_1 = jxcp_s->PROFINET_Mapping_IN.Input_Area[1];
				// Calculation Boolean (True/False) array (Byte 1)
				for(i = 0; i < (int)(sizeof(jxcp_s->Internal.Profinet.OUT_Aux.BYTE_1)/sizeof(jxcp_s->Internal.Profinet.OUT_Aux.BYTE_1[0])); i++){
					if(aux_get_byte_1 > 0){
						jxcp_s->Internal.Profinet.OUT_Aux.BYTE_1[i] = aux_get_byte_1 % 2;
						aux_get_byte_1 = aux_get_byte_1/2;
					}else{
						jxcp_s->Internal.Profinet.OUT_Aux.BYTE_1[i] = 0;
					}
				}

				// *************** Byte 2 *************** //
				// Read Profinet Var. -> Set Bool
				if(jxcp_s->PROFINET_Mapping_IN.Input_Area[2] == 16){
					jxcp_s->Internal.Profinet.OUT_Aux.BYTE_2 = 1;
				}else{
					jxcp_s->Internal.Profinet.OUT_Aux.BYTE_2 = 0;
				}

				// *************** Current Position *************** //
				// Number of Variables (USINT)
				m_u2d_cP.Count_of_VAR = 4;
				// Read -> PROFINET Var.
				m_u2d_cP.USINT_1 = jxcp_s->PROFINET_Mapping_IN.Input_Area[4];
				m_u2d_cP.USINT_2 = jxcp_s->PROFINET_Mapping_IN.Input_Area[5];
				m_u2d_cP.USINT_3 = jxcp_s->PROFINET_Mapping_IN.Input_Area[6];
				m_u2d_cP.USINT_4 = jxcp_s->PROFINET_Mapping_IN.Input_Area[7];
				// Call Function Block (Multiple USINT to Decimal)
				multiple_usint_to_dec(&m_u2d_cP);
				// Result (Decimal Variable)
				jxcp_s->Output.Current_Position = m_u2d_cP.Result_Decimal;

				// *************** Current Speed *************** //
				// Number of Variables (USINT)
				m_u2d_cS.Count_of_VAR = 2;
				// Read -> PROFINET Var.
				m_u2d_cS.USINT_1 = jxcp_s->PROFINET_Mapping_IN.Input_Area[8];
				m_u2d_cS.USINT_2 = jxcp_s->PROFINET_Mapping_IN.Input_Area[9];
				// Call Function Block (Multiple USINT to Decimal)
				multiple_usint_to_dec(&m_u2d_cS);
				// Result (Decimal Variable)
				jxcp_s->Output.Current_Speed = m_u2d_cS.Result_Decimal;

				// *************** Current Pushing Force *************** //
				// Number of Variables (USINT)
				m_u2d_cPF.Count_of_VAR = 2;
				// Read -> PROFINET Var.
				m_u2d_cPF.USINT_1 = jxcp_s->PROFINET_Mapping_IN.Input_Area[10];
				m_u2d_cPF.USINT_2 = jxcp_s->PROFINET_Mapping_IN.Input_Area[11];
				// Call Function Block (Multiple USINT to Decimal)
				multiple_usint_to_dec(&m_u2d_cPF);
				// Result (Decimal Variable)
				jxcp_s->Output.Current_Pushing_Force = m_u2d_cPF.Result_Decimal;

				// *************** Target Position *************** //
				// Number of Variables (USINT)
				m_u2d_TP.Count_of_VAR = 4;
				// Read -> PROFINET Var.
				m_u2d_TP.USINT_1 = jxcp_s->PROFINET_Mapping_IN.Input_Area[12];
				m_u2d_TP.USINT_2 = jxcp_s->PROFINET_Mapping_IN.Input_Area[13];
				m_u2d_TP.USINT_3 = jxcp_s->PROFINET_Mapping_IN.Input_Area[14];
				m_u2d_TP.USINT_4 = jxcp_s->PROFINET_Mapping_IN.Input_Area[15];
				// Call Function Block (Multiple USINT to Decimal)
				multiple_usint_to_dec(&m_u2d_TP);
				// Result (Decimal Variable)
				jxcp_s->Output.Target_Position = m_u2d_TP.Result_Decimal;

				// *************** Byte 16 - 19 {ALARM} *************** //
				// Read -> PROFINET Var.
				jxcp_s->Output.Warning.Alarm_1 = jxcp_s->PROFINET_Mapping_IN.Input_Area[16];
				// Read -> PROFINET Var.
				jxcp_s->Output.Warning.Alarm_2 = jxcp_s->PROFINET_Mapping_IN.Input_Area[17];
				// Read -> PROFINET Var.
				jxcp_s->Output.Warning.Alarm_3 = jxcp_s->PROFINET_Mapping_IN.Input_Area[18];
				// Read -> PROFINET Var.
				jxcp_s->Output.Warning.Alarm_4 = jxcp_s->PROFINET_Mapping_IN.Input_Area[19];

				// ************************************************************************ //
				// ********************************* WRITE ******************************** //
				// ************************************************************************ //

				// *************** Byte 0 *************** //
				// Create aux. variable
				USINT aux_set_byte_0;
				// Initialization
				aux_set_byte_0 = 0;
				// Calculation from Boolean (True/False) -> USINT (Byte 0)
				for(i = 0; i < (int)(sizeof(jxcp_s->Internal.Profinet.IN_Aux.BYTE_0)/sizeof(jxcp_s->Internal.Profinet.IN_Aux.BYTE_0[0])); i++){
					if(jxcp_s->Internal.Profinet.IN_Aux.BYTE_0[i] == 1){
						aux_set_byte_0 += pow(2, i);
					}
				}
				// Result Profinet (USINT)
				jxcp_s->PROFINET_Mapping_OUT.Output_Area[0] = aux_set_byte_0;

				// *************** Byte 1 *************** //
				// Create aux. variable
				USINT aux_set_byte_1;
				// Initialization
				aux_set_byte_1 = 0;
				// Calculation from Boolean (True/False) -> USINT (Byte 1)
				for(i = 0; i < (int)(sizeof(jxcp_s->Internal.Profinet.IN_Aux.BYTE_1)/sizeof(jxcp_s->Internal.Profinet.IN_Aux.BYTE_1[0])); i++){
					if(jxcp_s->Internal.Profinet.IN_Aux.BYTE_1[i] == 1){
						aux_set_byte_1 += pow(2, i);
					}
				}
				// Result Profinet (USINT)
				jxcp_s->PROFINET_Mapping_OUT.Output_Area[1] = aux_set_byte_1;

				// *************** Byte 2 *************** //
				// Create aux. variable
				USINT aux_set_byte_2;
				// Initialization
				aux_set_byte_2 = 0;
				// Calculation from Boolean (True/False) -> USINT (Byte 2)
				for(i = 0; i < (int)(sizeof(jxcp_s->Internal.Profinet.IN_Aux.BYTE_2)/sizeof(jxcp_s->Internal.Profinet.IN_Aux.BYTE_2[0])); i++){
					if(jxcp_s->Internal.Profinet.IN_Aux.BYTE_2[i] == 1){
						aux_set_byte_2 += pow(2, i);
					}
				}
				// Result Profinet (USINT)
				jxcp_s->PROFINET_Mapping_OUT.Output_Area[2] = aux_set_byte_2;

				// *************** Byte 3 *************** //
				// Create aux. variable
				USINT aux_set_byte_3;
				// Initialization
				aux_set_byte_3 = 0;

				for(i = 0; i < (int)(sizeof(jxcp_s->Internal.Profinet.IN_Aux.BYTE_3)/sizeof(jxcp_s->Internal.Profinet.IN_Aux.BYTE_3[0])); i++){
					if(jxcp_s->Internal.Profinet.IN_Aux.BYTE_3[i] == 1){
						aux_set_byte_3 += pow(2, i);
					}
				}
				// Result Profinet (USINT)
				jxcp_s->PROFINET_Mapping_OUT.Output_Area[3] = aux_set_byte_3;

				// *************** Byte 4 *************** //
				// Write Profinet Var. -> Set USINT
				if(jxcp_s->Input.Start_Flag == 1){
					jxcp_s->PROFINET_Mapping_OUT.Output_Area[4] = 1;
				}else{
					jxcp_s->PROFINET_Mapping_OUT.Output_Area[4] = 0;
				}
				// *************** Byte 5 *************** //
				// Write Profinet Var. -> Set USINT
				if(jxcp_s->Input.Movement_Mode.Absolute == 1){
					// Movement -> Absolute
					jxcp_s->PROFINET_Mapping_OUT.Output_Area[5] = 1;
				}else if(jxcp_s->Input.Movement_Mode.Relative == 1){
					// Movement -> Relative
					jxcp_s->PROFINET_Mapping_OUT.Output_Area[5] = 2;
				}else{
					// Movement -> NULL
					jxcp_s->PROFINET_Mapping_OUT.Output_Area[5] = 0;
				}

				// Module OK = 0 -> Error State
				if(jxcp_s->ModuleOK != 1){
					// Set FB -> Active 0
					jxcp_s->Active = 0;
					// Change State -> Error
					jxcp_s->Internal.actual_r_state = JXCP_R_ERROR_MODE_STATE;
				}
			}
			break;
		case JXCP_R_ERROR_MODE_STATE:
			{
				/*************************************** ERROR STATE ******************************************/
				// Profinet Module -> OK
				if(jxcp_s->ModuleOK == 1){
					// Set FB -> Active 1
					jxcp_s->Active = 1;
					// Change State -> before state (before the error)
					jxcp_s->Internal.actual_r_state = jxcp_s->Internal.before_r_state;
				}
			}
			break;
	} // end switch

	/*************************************** R/W DATA ******************************************/
	if(jxcp_s->Active == 1){
		// Read Data {Transform Single Data -> ARRAY}
		// Byte 0 {INPUT}
		jxcp_s->Internal.Profinet.IN_Aux.BYTE_0[0] = jxcp_s->Input.BYTE_0.IN_0;
		jxcp_s->Internal.Profinet.IN_Aux.BYTE_0[1] = jxcp_s->Input.BYTE_0.IN_1;
		jxcp_s->Internal.Profinet.IN_Aux.BYTE_0[2] = jxcp_s->Input.BYTE_0.IN_2;
		jxcp_s->Internal.Profinet.IN_Aux.BYTE_0[3] = jxcp_s->Input.BYTE_0.IN_3;
		jxcp_s->Internal.Profinet.IN_Aux.BYTE_0[4] = jxcp_s->Input.BYTE_0.IN_4;
		jxcp_s->Internal.Profinet.IN_Aux.BYTE_0[5] = jxcp_s->Input.BYTE_0.IN_5;
		// Byte 1 {INPUT}
		jxcp_s->Internal.Profinet.IN_Aux.BYTE_1[0] = jxcp_s->Input.BYTE_1.HOLD;
		jxcp_s->Internal.Profinet.IN_Aux.BYTE_1[1] = jxcp_s->Input.BYTE_1.SVON;
		jxcp_s->Internal.Profinet.IN_Aux.BYTE_1[2] = jxcp_s->Input.BYTE_1.DRIVE;
		jxcp_s->Internal.Profinet.IN_Aux.BYTE_1[3] = jxcp_s->Input.BYTE_1.RESET;
		jxcp_s->Internal.Profinet.IN_Aux.BYTE_1[4] = jxcp_s->Input.BYTE_1.SETUP;
		jxcp_s->Internal.Profinet.IN_Aux.BYTE_1[5] = jxcp_s->Input.BYTE_1.JOG_Neg;
		jxcp_s->Internal.Profinet.IN_Aux.BYTE_1[6] = jxcp_s->Input.BYTE_1.JOG_Pos;
		jxcp_s->Internal.Profinet.IN_Aux.BYTE_1[7] = jxcp_s->Input.BYTE_1.FLHGT;
		// Byte 2 {INPUT}
		jxcp_s->Internal.Profinet.IN_Aux.BYTE_2[0] = 0;
		jxcp_s->Internal.Profinet.IN_Aux.BYTE_2[1] = jxcp_s->Input.BYTE_2.Speed_Restriction;
		jxcp_s->Internal.Profinet.IN_Aux.BYTE_2[2] = 0;
		jxcp_s->Internal.Profinet.IN_Aux.BYTE_2[3] = 0;
		jxcp_s->Internal.Profinet.IN_Aux.BYTE_2[4] = jxcp_s->Input.BYTE_2.Movement_Mode;
		jxcp_s->Internal.Profinet.IN_Aux.BYTE_2[5] = jxcp_s->Input.BYTE_2.Speed;
		jxcp_s->Internal.Profinet.IN_Aux.BYTE_2[6] = jxcp_s->Input.BYTE_2.Position;
		jxcp_s->Internal.Profinet.IN_Aux.BYTE_2[7] = jxcp_s->Input.BYTE_2.Acceleration;
		// Byte 3 {INPUT}
		jxcp_s->Internal.Profinet.IN_Aux.BYTE_3[0] = jxcp_s->Input.BYTE_3.Deceleration;
		jxcp_s->Internal.Profinet.IN_Aux.BYTE_3[1] = jxcp_s->Input.BYTE_3.Pushing_Force;
		jxcp_s->Internal.Profinet.IN_Aux.BYTE_3[2] = jxcp_s->Input.BYTE_3.Trigger_LV;
		jxcp_s->Internal.Profinet.IN_Aux.BYTE_3[3] = jxcp_s->Input.BYTE_3.Pushing_Speed;
		jxcp_s->Internal.Profinet.IN_Aux.BYTE_3[4] = jxcp_s->Input.BYTE_3.Moving_Force;
		jxcp_s->Internal.Profinet.IN_Aux.BYTE_3[5] = jxcp_s->Input.BYTE_3.Area_out_1;
		jxcp_s->Internal.Profinet.IN_Aux.BYTE_3[6] = jxcp_s->Input.BYTE_3.Area_out_2;
		jxcp_s->Internal.Profinet.IN_Aux.BYTE_3[7] = jxcp_s->Input.BYTE_3.IN_Pos_Tolerance;
		// Write Data {Transform ARRAY -> Single Data}
		// Byte 0 {OUTPUT}
		jxcp_s->Output.BYTE_0.OUT_0 = jxcp_s->Internal.Profinet.OUT_Aux.BYTE_0[0];
		jxcp_s->Output.BYTE_0.OUT_1 = jxcp_s->Internal.Profinet.OUT_Aux.BYTE_0[1];
		jxcp_s->Output.BYTE_0.OUT_2 = jxcp_s->Internal.Profinet.OUT_Aux.BYTE_0[2];
		jxcp_s->Output.BYTE_0.OUT_3 = jxcp_s->Internal.Profinet.OUT_Aux.BYTE_0[3];
		jxcp_s->Output.BYTE_0.OUT_4 = jxcp_s->Internal.Profinet.OUT_Aux.BYTE_0[4];
		jxcp_s->Output.BYTE_0.OUT_5 = jxcp_s->Internal.Profinet.OUT_Aux.BYTE_0[5];
		// Byte 1 {OUTPUT}
		jxcp_s->Output.BYTE_1.BUSY  = jxcp_s->Internal.Profinet.OUT_Aux.BYTE_1[0];
		jxcp_s->Output.BYTE_1.SVRE  = jxcp_s->Internal.Profinet.OUT_Aux.BYTE_1[1];
		jxcp_s->Output.BYTE_1.SETON = jxcp_s->Internal.Profinet.OUT_Aux.BYTE_1[2];
		jxcp_s->Output.BYTE_1.INP   = jxcp_s->Internal.Profinet.OUT_Aux.BYTE_1[3];
		jxcp_s->Output.BYTE_1.AREA  = jxcp_s->Internal.Profinet.OUT_Aux.BYTE_1[4];
		jxcp_s->Output.BYTE_1.WAREA = jxcp_s->Internal.Profinet.OUT_Aux.BYTE_1[5];
		jxcp_s->Output.BYTE_1.ESTOP = jxcp_s->Internal.Profinet.OUT_Aux.BYTE_1[6];
		jxcp_s->Output.BYTE_1.ALARM = jxcp_s->Internal.Profinet.OUT_Aux.BYTE_1[7];
		// Byte 2 {OUTPUT}
		jxcp_s->Output.BYTE_2.READY = jxcp_s->Internal.Profinet.OUT_Aux.BYTE_2;

	}
} // end function block

// ************************************************************************************************************************************ //
// ------------------------------------------------------------  FUNCTIONS ------------------------------------------------------------ //
// ************************************************************************************************************************************ //

// ****************INITIALIZATION PARAMETERS ********************** //
void initialization_jxcp(struct jxcp_smc_fb* jxcp_s)
{
	// Initialization state {Main JXCP}
	jxcp_s->Internal.actual_state = JXCP_INITIALIZATION_STATE;
	jxcp_s->Internal.before_state = JXCP_INITIALIZATION_STATE;
	// Initialization state {READ/Write JXCP}
	jxcp_s->Internal.actual_r_state = JXCP_R_INITIALIZATION_STATE;
	jxcp_s->Internal.before_r_state = JXCP_R_INITIALIZATION_STATE;
	// Set Parameters
	// Mode
	jxcp_s->Set_Parameters.Mode = NORMAL_MOVE_MODE;
	// Start/Stop
	jxcp_s->Set_Parameters.Start = 0;
	jxcp_s->Set_Parameters.Stop  = 0;
	// ----- INPUT (FB) ----- //
	// Input {Byte 0}
	jxcp_s->Input.BYTE_0.IN_0 = 0;
	jxcp_s->Input.BYTE_0.IN_1 = 0;
	jxcp_s->Input.BYTE_0.IN_2 = 0;
	jxcp_s->Input.BYTE_0.IN_3 = 0;
	jxcp_s->Input.BYTE_0.IN_4 = 0;
	jxcp_s->Input.BYTE_0.IN_5 = 0;
	// Input {Byte 1}
	jxcp_s->Input.BYTE_1.DRIVE   = 0;
	jxcp_s->Input.BYTE_1.FLHGT   = 0;
	jxcp_s->Input.BYTE_1.HOLD    = 0;
	jxcp_s->Input.BYTE_1.JOG_Neg = 0;
	jxcp_s->Input.BYTE_1.JOG_Pos = 0;
	jxcp_s->Input.BYTE_1.RESET   = 0;
	jxcp_s->Input.BYTE_1.SETUP   = 0;
	jxcp_s->Input.BYTE_1.SVON    = 0;
	// Input {Byte 2}
	jxcp_s->Input.BYTE_2.Acceleration      = 0;
	jxcp_s->Input.BYTE_2.Movement_Mode     = 0;
	jxcp_s->Input.BYTE_2.Position          = 0;
	jxcp_s->Input.BYTE_2.Speed             = 0;
	jxcp_s->Input.BYTE_2.Speed_Restriction = 0;
	// Input {Byte 3}
	jxcp_s->Input.BYTE_3.Area_out_1       = 0;
	jxcp_s->Input.BYTE_3.Area_out_2       = 0;
	jxcp_s->Input.BYTE_3.Deceleration     = 0;
	jxcp_s->Input.BYTE_3.IN_Pos_Tolerance = 0;
	jxcp_s->Input.BYTE_3.Moving_Force     = 0;
	jxcp_s->Input.BYTE_3.Pushing_Force    = 0;
	jxcp_s->Input.BYTE_3.Pushing_Speed    = 0;
	jxcp_s->Input.BYTE_3.Trigger_LV       = 0;
	// Input {Byte 4}
	jxcp_s->Input.Start_Flag = 0;
	// Input {Byte 5}
	jxcp_s->Input.Movement_Mode.Absolute = 0;
	jxcp_s->Input.Movement_Mode.Relative = 0;
	// Input {Byte 6 - 7}
	jxcp_s->Input.Speed = 0;
	// Input {Byte 8 - 11}
	jxcp_s->Input.Position = 0;
	// Input {Byte 12 - 13}
	jxcp_s->Input.Acceleration = 0;
	// Input {Byte 14 - 15}
	jxcp_s->Input.Deceleration = 0;
	// Input {Byte 16 - 17}
	jxcp_s->Input.Pushing_Force = 0;
	// Input {Byte 18 - 19}
	jxcp_s->Input.Trigger_LV = 0;
	// Input {Byte 20 - 21}
	jxcp_s->Input.Pushing_Speed = 0;
	// Input {Byte 22 - 23}
	jxcp_s->Input.Moving_Force = 0;
	// Input {Byte 24 - 27}
	jxcp_s->Input.AREA_1 = 0;
	// Input {Byte 28 - 31}
	jxcp_s->Input.AREA_2 = 0;
	// Input {Byte 32 - 35}
	jxcp_s->Input.IN_Position = 0;
	// ----- INPUT (FB) ----- //
	// FB -> Active
	jxcp_s->Active = 0;
	// Output {Byte 0}
	jxcp_s->Output.BYTE_0.OUT_0 = 0;
	jxcp_s->Output.BYTE_0.OUT_1 = 0;
	jxcp_s->Output.BYTE_0.OUT_2 = 0;
	jxcp_s->Output.BYTE_0.OUT_3 = 0;
	jxcp_s->Output.BYTE_0.OUT_4 = 0;
	jxcp_s->Output.BYTE_0.OUT_5 = 0;
	// Output {Byte 1}
	jxcp_s->Output.BYTE_1.ALARM = 0;
	jxcp_s->Output.BYTE_1.AREA  = 0;
	jxcp_s->Output.BYTE_1.BUSY  = 0;
	jxcp_s->Output.BYTE_1.ESTOP = 0;
	jxcp_s->Output.BYTE_1.INP   = 0;
	jxcp_s->Output.BYTE_1.SETON = 0;
	jxcp_s->Output.BYTE_1.SVRE  = 0;
	jxcp_s->Output.BYTE_1.WAREA = 0;
	// Output {Byte 2}
	jxcp_s->Output.BYTE_2.READY = 0;
	// Output {Byte 4 - 7}
	jxcp_s->Output.Current_Position = 0;
	// Output {Byte 8 - 9}
	jxcp_s->Output.Current_Speed = 0;
	// Output {Byte 10 - 11}
	jxcp_s->Output.Current_Pushing_Force = 0;
	// Output {Byte 12 - 15}
	jxcp_s->Output.Target_Position = 0;
	// Output {Byte 16}
	jxcp_s->Output.Warning.Alarm_1 = 0;
	// Output {Byte 17}
	jxcp_s->Output.Warning.Alarm_2 = 0;
	// Output {Byte 18}
	jxcp_s->Output.Warning.Alarm_3 = 0;
	// Output {Byte 19}
	jxcp_s->Output.Warning.Alarm_4 = 0;
	// Output -> PROFINET {Byte 0 - 35}
	jxcp_s->PROFINET_Mapping_OUT.Output_Area[0] = 0;
	jxcp_s->PROFINET_Mapping_OUT.Output_Area[1] = 0;
	jxcp_s->PROFINET_Mapping_OUT.Output_Area[2] = 0;
	jxcp_s->PROFINET_Mapping_OUT.Output_Area[3] = 0;
	jxcp_s->PROFINET_Mapping_OUT.Output_Area[4] = 0;
	jxcp_s->PROFINET_Mapping_OUT.Output_Area[5] = 0;
	jxcp_s->PROFINET_Mapping_OUT.Output_Area[6] = 0;
	jxcp_s->PROFINET_Mapping_OUT.Output_Area[7] = 0;
	jxcp_s->PROFINET_Mapping_OUT.Output_Area[8] = 0;
	jxcp_s->PROFINET_Mapping_OUT.Output_Area[9] = 0;
	jxcp_s->PROFINET_Mapping_OUT.Output_Area[10] = 0;
	jxcp_s->PROFINET_Mapping_OUT.Output_Area[11] = 0;
	jxcp_s->PROFINET_Mapping_OUT.Output_Area[12] = 0;
	jxcp_s->PROFINET_Mapping_OUT.Output_Area[13] = 0;
	jxcp_s->PROFINET_Mapping_OUT.Output_Area[14] = 0;
	jxcp_s->PROFINET_Mapping_OUT.Output_Area[15] = 0;
	jxcp_s->PROFINET_Mapping_OUT.Output_Area[16] = 0;
	jxcp_s->PROFINET_Mapping_OUT.Output_Area[17] = 0;
	jxcp_s->PROFINET_Mapping_OUT.Output_Area[18] = 0;
	jxcp_s->PROFINET_Mapping_OUT.Output_Area[19] = 0;
	jxcp_s->PROFINET_Mapping_OUT.Output_Area[20] = 0;
	jxcp_s->PROFINET_Mapping_OUT.Output_Area[21] = 0;
	jxcp_s->PROFINET_Mapping_OUT.Output_Area[22] = 0;
	jxcp_s->PROFINET_Mapping_OUT.Output_Area[23] = 0;
	jxcp_s->PROFINET_Mapping_OUT.Output_Area[24] = 0;
	jxcp_s->PROFINET_Mapping_OUT.Output_Area[25] = 0;
	jxcp_s->PROFINET_Mapping_OUT.Output_Area[26] = 0;
	jxcp_s->PROFINET_Mapping_OUT.Output_Area[27] = 0;
	jxcp_s->PROFINET_Mapping_OUT.Output_Area[28] = 0;
	jxcp_s->PROFINET_Mapping_OUT.Output_Area[29] = 0;
	jxcp_s->PROFINET_Mapping_OUT.Output_Area[30] = 0;
	jxcp_s->PROFINET_Mapping_OUT.Output_Area[31] = 0;
	jxcp_s->PROFINET_Mapping_OUT.Output_Area[32] = 0;
	jxcp_s->PROFINET_Mapping_OUT.Output_Area[33] = 0;
	jxcp_s->PROFINET_Mapping_OUT.Output_Area[34] = 0;
	jxcp_s->PROFINET_Mapping_OUT.Output_Area[35] = 0;
} // end function

// **************** MULTIPLE USINT TO DECIMAL ********************** //
void multiple_usint_to_dec(struct multiple_usint_to_dec* m_u2d){

	// Declaration {2 - variables}
	// Index
	int i_2;
	// Aux. array -> result
	int result_bin_byte_2[16];
	int result_bin_byte_21[8], result_bin_byte_22[8];
	// Aux. USINT
	USINT aux_get_byte_21, aux_get_byte_22;
	// Initialization
	LREAL aux_set_dec_2 = 0;
	// Array size
	int n_2 = (int)(sizeof(result_bin_byte_2)/sizeof(result_bin_byte_2[0]));

	// Declaration {4 - variables}
	// Index
	int i_4;
	// Aux. array -> result
	int result_bin_byte_4[32];
	int result_bin_byte_41[8], result_bin_byte_42[8], result_bin_byte_43[8], result_bin_byte_44[8];
	// Aux. USINT
	USINT aux_get_byte_41, aux_get_byte_42, aux_get_byte_43, aux_get_byte_44;
	// Initialization
	LREAL aux_set_dec_4 = 0;
	// Array size
	int n_4 = (int)(sizeof(result_bin_byte_4)/sizeof(result_bin_byte_4[0]));

	// ************************************************************************ //
	// --------------------------- MAIN STATE --------------------------------- //
	// ************************************************************************ //
	switch(m_u2d->Count_of_VAR){
		case 2:
			{
				// ********************************** Variables 2 ************************************** //
				// INPUT {USINT}
				aux_get_byte_21 = m_u2d->USINT_1;
				aux_get_byte_22 = m_u2d->USINT_2;

				// ********** Calculation ********** //
				for(i_2 = 0; i_2 < (int)(sizeof(result_bin_byte_21)/sizeof(result_bin_byte_21[0])); i_2++){
					// USINT 1 -> Boolean Array
					if(aux_get_byte_21 > 0){
						result_bin_byte_21[i_2] = fmod(aux_get_byte_21, 2);
						aux_get_byte_21 = aux_get_byte_21/2;
					}else{
						result_bin_byte_21[i_2] = 0;
					}
					// USINT 2 -> Boolean Array
					if(aux_get_byte_22 > 0){
						result_bin_byte_22[i_2] = fmod(aux_get_byte_22, 2);
						aux_get_byte_22 = aux_get_byte_22/2;
					}else{
						result_bin_byte_22[i_2] = 0;
					}
				}

				// Create a single array from multiple USINT  -> {USINT 1, USINT 2}
				for(i_2 = 0; i_2 < n_2; i_2++){
					if(i_2 >= 0 && i_2 < 8){
						result_bin_byte_2[i_2] = result_bin_byte_22[i_2];
					}else if(i_2 >= 8 && i_2 < 16){
						result_bin_byte_2[i_2] = result_bin_byte_21[i_2 - 8];
					}
				}

				// Create LREAL number
				for(i_2 = 0; i_2 < n_2; i_2++){
					if(result_bin_byte_2[i_2] == 1){
						aux_set_dec_2 = aux_set_dec_2 + pow(10, i_2);
					}
				}

				// Result -> Decimal Number
				m_u2d->Result_Decimal = (LREAL)convert_bin_to_dec(aux_set_dec_2);
			}
			break;
		case 4:
			{
				// ********************************** Variables 4 ************************************** //
				// INPUT {USINT}
				aux_get_byte_41 = m_u2d->USINT_1;
				aux_get_byte_42 = m_u2d->USINT_2;
				aux_get_byte_43 = m_u2d->USINT_3;
				aux_get_byte_44 = m_u2d->USINT_4;

				// ********** Calculation ********** //
				for(i_4 = 0; i_4 < (int)(sizeof(result_bin_byte_41)/sizeof(result_bin_byte_41[0])); i_4++){
					// USINT 1 -> Boolean Array
					if(aux_get_byte_41 > 0){
						result_bin_byte_41[i_4] = fmod(aux_get_byte_41, 2);
						aux_get_byte_41 = aux_get_byte_41/2;
					}else{
						result_bin_byte_41[i_4] = 0;
					}
					// USINT 2 -> Boolean Array
					if(aux_get_byte_42 > 0){
						result_bin_byte_42[i_4] = fmod(aux_get_byte_42, 2);
						aux_get_byte_42 = aux_get_byte_42/2;
					}else{
						result_bin_byte_42[i_4] = 0;
					}
					// USINT 3 -> Boolean Array
					if(aux_get_byte_43 > 0){
						result_bin_byte_43[i_4] = fmod(aux_get_byte_43, 2);
						aux_get_byte_43 = aux_get_byte_43/2;
					}else{
						result_bin_byte_43[i_4] = 0;
					}
					// USINT 4 -> Boolean Array
					if(aux_get_byte_44 > 0){
						result_bin_byte_44[i_4] = fmod(aux_get_byte_44, 2);
						aux_get_byte_44 = aux_get_byte_44/2;
					}else{
						result_bin_byte_44[i_4] = 0;
					}
				}

				// Create a single array from multiple USINT -> {USINT 1, USINT 2, USINT 3, USINT 4}
				for(i_4 = 0; i_4 < n_4; i_4++){
					if(i_4 >= 0 && i_4 < 8){
						result_bin_byte_4[i_4] = result_bin_byte_44[i_4];
					}else if(i_4 >= 8 && i_4 < 16){
						result_bin_byte_4[i_4] = result_bin_byte_43[i_4 - 8];
					}else if(i_4 >= 16 && i_4 < 24){
						result_bin_byte_4[i_4] = result_bin_byte_42[i_4 - 16];
					}else if(i_4 >= 24 && i_4 < 32){
						result_bin_byte_4[i_4] = result_bin_byte_41[i_4 - 24];
					}
				}

				// Create LREAL number
				for(i_4 = 0; i_4 < n_4; i_4++){
					if(result_bin_byte_4[i_4] == 1){
						aux_set_dec_4 = aux_set_dec_4 + pow(10,i_4);
					}
				}

				// Result -> Decimal Number
				m_u2d->Result_Decimal = ((LREAL)convert_bin_to_dec(aux_set_dec_4))*0.01;
			}
			break;
	}
} // end function

// **************** DECIMAL TO MULTIPLE USINT ********************** //
void dec_to_multiple_usint(struct dec_to_multiple_usint* dec2u_m){

	// Declaration {2 - variables}
	// Index
	int i_2;
	// Aux. array -> result
	int result_bin_byte_2[16];
	int result_bin_byte_21[8], result_bin_byte_22[8];
	// Aux. USINT
	LREAL aux_get_dec_2;
	// Initialization
	USINT aux_set_byte_21 = 0, aux_set_byte_22 = 0;
	// Array size
	int n_2 = (int)(sizeof(result_bin_byte_2)/sizeof(result_bin_byte_2[0]));

	// Declaration {4 - variables}
	// Index
	int i_4;
	// Aux. array -> result
	int result_bin_byte_4[32];
	int result_bin_byte_41[8], result_bin_byte_42[8], result_bin_byte_43[8], result_bin_byte_44[8];
	// Aux. USINT
	LREAL aux_get_dec_4;
	// Initialization
	USINT aux_set_byte_41 = 0, aux_set_byte_42 = 0, aux_set_byte_43 = 0, aux_set_byte_44 = 0;
	// Array size
	int n_4 = (int)(sizeof(result_bin_byte_4)/sizeof(result_bin_byte_4[0]));

	// ************************************************************************ //
	// --------------------------- MAIN STATE --------------------------------- //
	// ************************************************************************ //
	switch(dec2u_m->Count_of_VAR){
		case 2:
			{
				// ********************************** Variables 2 ************************************** //
				// INPUT {DECIMAL}
				aux_get_dec_2 = dec2u_m->Decimal;

				// ********** Calculation {Array} ********** //
				// Transform decimal to boolean (true/false) array
				for(i_2 = 0; i_2 < n_2; i_2++){
					result_bin_byte_2[i_2] = fmod(aux_get_dec_2, 2);
					aux_get_dec_2		   = aux_get_dec_2/2;
				}

				// Create multiple separate array
				for(i_2 = 0; i_2 < n_2; i_2++){
					if(i_2 >= 0 && i_2 < 8){
						result_bin_byte_22[i_2]      = result_bin_byte_2[i_2];
					}else if(i_2 >= 8 && i_2 < 16){
						result_bin_byte_21[i_2 - 8]  = result_bin_byte_2[i_2];
					}
				}

				// ********** Calculation {USINT} ********** //
				for(i_2 = 0; i_2 < (int)(sizeof(result_bin_byte_21)/sizeof(result_bin_byte_21[0])); i_2++){
					// USINT 1
					if(result_bin_byte_21[i_2] == 1){
						aux_set_byte_21 += pow(2, i_2);
					}
					// USINT 2
					if(result_bin_byte_22[i_2] == 1){
						aux_set_byte_22 += pow(2, i_2);
					}
				}

				// Result -> Multiple USINT
				dec2u_m->Result_USINT_1 = aux_set_byte_21;
				dec2u_m->Result_USINT_2 = aux_set_byte_22;
			}
			break;
		case 4:
			{
				// ********************************** Variables 4 ************************************** //
				// INPUT {DECIMAL}
				aux_get_dec_4 = dec2u_m->Decimal * 100;

				// ********** Calculation {Array} ********** //
				// Transform decimal to boolean (true/false) array
				for(i_4 = 0; i_4 < n_4; i_4++){
					result_bin_byte_4[i_4] = fmod(aux_get_dec_4, 2);
					aux_get_dec_4		   = aux_get_dec_4/2;
				}

				// Create multiple separate array
				for(i_4 = 0; i_4 < n_4; i_4++){
					if(i_4 >= 0 && i_4 < 8){
						result_bin_byte_44[i_4]      = result_bin_byte_4[i_4];
					}else if(i_4 >= 8 && i_4 < 16){
						result_bin_byte_43[i_4 - 8]  = result_bin_byte_4[i_4];
					}else if(i_4 >= 16 && i_4 < 24){
						result_bin_byte_42[i_4 - 16] = result_bin_byte_4[i_4];
					}else if(i_4 >= 24 && i_4 < 32){
						result_bin_byte_41[i_4 - 24] = result_bin_byte_4[i_4];
					}
				}

				// ********** Calculation {USINT} ********** //
				for(i_4 = 0; i_4 < (int)(sizeof(result_bin_byte_41)/sizeof(result_bin_byte_41[0])); i_4++){
					// USINT 1
					if(result_bin_byte_41[i_4] == 1){
						aux_set_byte_41 += pow(2, i_4);
					}
					// USINT 2
					if(result_bin_byte_42[i_4] == 1){
						aux_set_byte_42 += pow(2, i_4);
					}
					// USINT 3
					if(result_bin_byte_43[i_4] == 1){
						aux_set_byte_43 += pow(2, i_4);
					}
					// USINT 4
					if(result_bin_byte_44[i_4] == 1){
						aux_set_byte_44 += pow(2, i_4);
					}
				}

				// Result -> Multiple USINT
				dec2u_m->Result_USINT_1 = aux_set_byte_41;
				dec2u_m->Result_USINT_2 = aux_set_byte_42;
				dec2u_m->Result_USINT_3 = aux_set_byte_43;
				dec2u_m->Result_USINT_4 = aux_set_byte_44;
			}
			break;
	}
} // end function

// **************** AUX. BINARY TO DECIMAL ********************** //
DINT convert_bin_to_dec(LREAL variable) {
	// initialization aux. variables
	DINT decimal_num = 0, i = 0, remainder;

	// calculation {binary -> decimal}
	for(i = 0; variable > 0; i++)
	{
		remainder    = fmod(variable, 10);
		decimal_num += remainder * pow(2,i);
		variable    /= 10;
	}

	// return decimal number {result}
	return decimal_num;
} // end function
```

### Program Logical/Technology/JXCP_Test (ANSIC)

#### Main.c
```c
#include <bur/plctypes.h>
#include <stdio.h>
#include <stdlib.h>
#include <math.h>

#include "rp_funcx.h"

#ifdef _DEFAULT_INCLUDES
	#include <AsDefault.h>
#endif

_LOCAL struct jxcp_smc_fb jxcp_smc_fb_1;

void _INIT ProgramInit(void)
{

	//jxcp_smc_fb_1.Enable = 1;

	jxcp_smc_fb_1.Set_Parameters.Mode = CYCLE_MOVE_MODE;

	jxcp_smc_fb_1.Input.Speed 		 = 50;
	jxcp_smc_fb_1.Input.Acceleration = 1000;
	jxcp_smc_fb_1.Input.Deceleration = 1000;
	jxcp_smc_fb_1.Input.Moving_Force = 100;
	jxcp_smc_fb_1.Input.IN_Position  = 0.5;
}

void _CYCLIC ProgramCyclic(void)
{
	jxcp_smc_fb(&jxcp_smc_fb_1);
}
```

- Visualisation Logical/mappView (not shown)

Listed in the project but not available here: Logical/Libraries/rp_funcx/Constants.var
